Omron CX-Programmer project NewProject (CX-Programmer 9.75)

# PLC NewPLC1: CP1L M

## Global symbols (name address type ; comment)
0.00 BOOL  ; Start
0.01 BOOL  ; Stop
0.02 BOOL  ; Emergency
0.03 BOOL  ; Sensor-1
0.04 BOOL  ; Sensor-2
100.00 BOOL  ; Buzzer
100.01 BOOL  ; Conveyor-1
100.02 BOOL  ; Conveyor-2
W0.00 BOOL  ; Start
W0.01 BOOL  ; Stop

## Program NewProgram1 (cyclic task 0)

### Section Section1

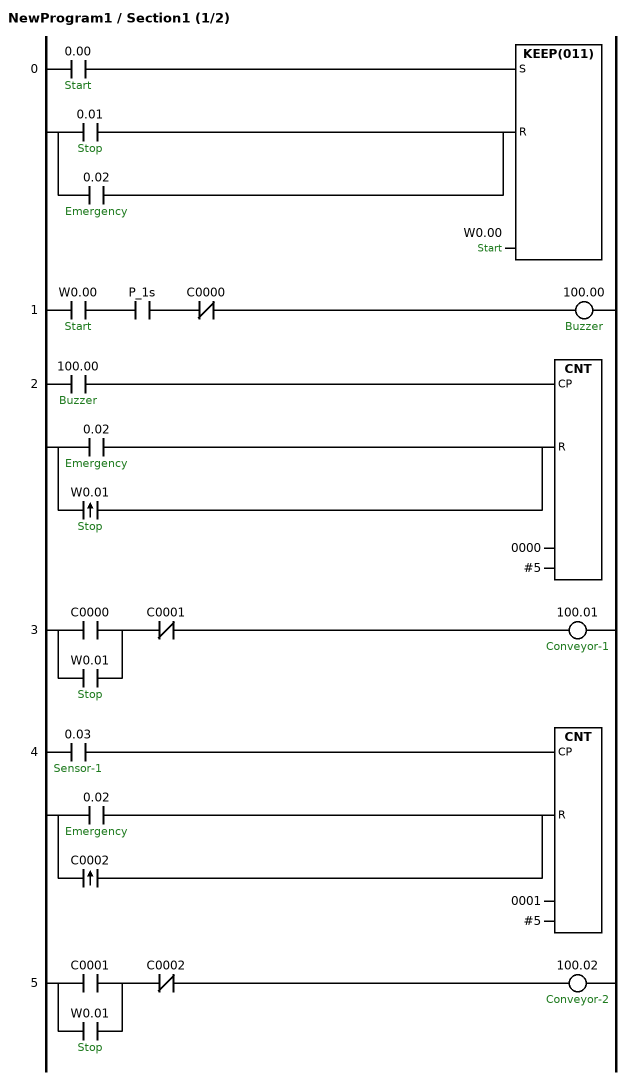
; rung 0
LD 0.00  ; Start
LD 0.01  ; Stop
OR 0.02  ; Emergency
KEEP(011) W0.00  ; Start
; rung 1
LD W0.00  ; Start
AND P_1s
ANDNOT C0000
OUT 100.00  ; Buzzer
; rung 2
LD 100.00  ; Buzzer
LD 0.02  ; Emergency
@OR W0.01  ; Stop
CNT 0000 #5
; rung 3
LD C0000
OR W0.01  ; Stop
ANDNOT C0001
OUT 100.01  ; Conveyor-1
; rung 4
LD 0.03  ; Sensor-1
LD 0.02  ; Emergency
@OR C0002
CNT 0001 #5
; rung 5
LD C0001
OR W0.01  ; Stop
ANDNOT C0002
OUT 100.02  ; Conveyor-2

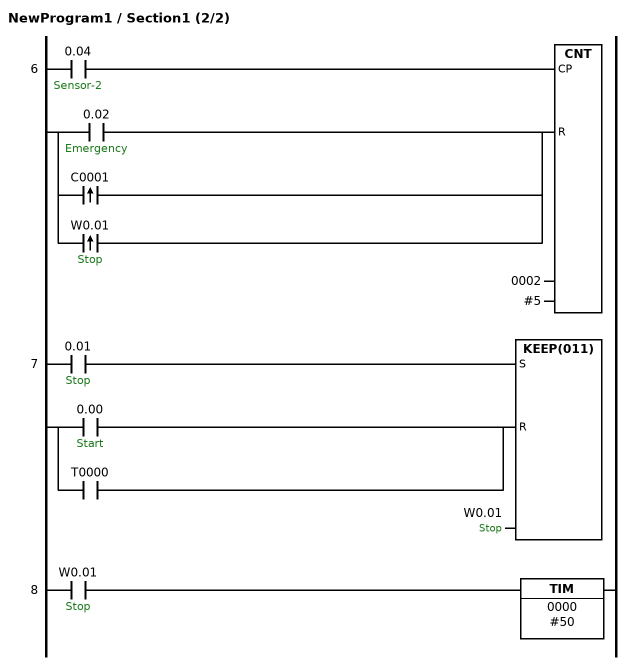
; rung 6
LD 0.04  ; Sensor-2
LD 0.02  ; Emergency
@OR C0001
@OR W0.01  ; Stop
CNT 0002 #5
; rung 7
LD 0.01  ; Stop
LD 0.00  ; Start
OR T0000
KEEP(011) W0.01  ; Stop
; rung 8
LD W0.01  ; Stop
TIM 0000 #50

### Section END
; rung 0
END(001)